			OR	NOT bSensAPVorhanden
			AND	NOT bE_sensRP
			AND		fbZeitAP.Q
			
			OR		bSensAPVorhanden
			AND NOT bSensRPVorhanden
			AND		bE_sensAP
			
			OR		bSensAPVorhanden
			AND		bE_sensAP
			AND NOT bE_sensRP) THEN
			
	eStatus := AktorStatus.inAP;
	
	IF			(eAnfrage = AktorStatus.zuAP) THEN
		bFalschePos := FALSE;
		eAnfrage := AktorStatus.default;
	END_IF

//http://www.32x8.com/sop6_____A-B-C-D-E-F_____m_1-3-5-7-10-11-14-15-17-19-26-27___________option-0_____989781966178824394701
ELSIF		NOT bA_arbeitsPos
		AND (NOT bSensAPVorhanden
		AND NOT bSensRPVorhanden
		AND		fbZeitRP.Q
		
		OR	NOT bSensRPVorhanden
		AND NOT bE_sensAP
		AND		fbZeitRP.Q
		
		OR	NOT bSensAPVorhanden
		AND		bSensRPVorhanden
		AND		bE_sensRP
		
		OR		bSensRPVorhanden
		AND NOT bE_sensAP
		AND		bE_sensRP) THEN
		
	eStatus := AktorStatus.inRP;
	
	IF			(eAnfrage = AktorStatus.zuRP) THEN
		bFalschePos := FALSE;
		eAnfrage := AktorStatus.default;
	END_IF
ELSE
	eStatus := AktorStatus.default;
END_IF

//Nothalt
IF		NOT	MAIN.bE_NotHalt THEN
	bArbeitsPos := FALSE;
	bFalschePos := FALSE;
END_IF

//Handbetrieb
IF			MAIN.bE_Handbetrieb THEN
	IF			bBtnHandausloesung THEN
		bBtnHandausloesung := FALSE;
		handAusloesung();
	END_IF
ELSE
	bBtnHandausloesung := FALSE;
END_IF

//Positionsüberwachung Handbetrieb
fbFtrigHandbetr(CLK := Main.bE_Handbetrieb);

IF 			(fbFtrigHandbetr.Q
	OR		fbSchrittbetrieb.bSendFalschePosError)
	AND		bFalschePos THEN
	
	IF			bA_arbeitsPos THEN
		EventLogger.aErrorLog[250].ipArguments.Clear().AddString(sBezeichnung).AddString('Ruheposition');
	ELSE
		EventLogger.aErrorLog[250].ipArguments.Clear().AddString(sBezeichnung).AddString('Arbeitsposition');
	END_IF
	
	EventLogger.aErrorLog[250].Send(0);
END_IF

IF 			bFalschePos THEN
	fbSchrittbetrieb.bAktorPosNIO := TRUE;
	Main.bPosNachHbNio := TRUE;
END_IF

METHOD arbeitsPos : BOOL
VAR_INPUT
END_VAR
VAR_INST
	bPrevOutputState: 		BOOL;
END_VAR
VAR
	stSchrittEintrag:		ST_SchrittQueue;
END_VAR
stSchrittEintrag.fbAktor REF= THIS^;	
stSchrittEintrag.bGesetzt := TRUE;

//*************************************************************************************
IF		NOT Main.bE_Handbetrieb 
	AND NOT Main.bProgStop
	OR		bHandOverride

	OR		MAIN.bE_Handbetrieb							//Schritt vorwaerts im Handbetrieb
	AND		fbSchrittbetrieb.bAblaufFreigabe THEN
	
	//*************************************************************************************
	IF		NOT bArbeitsPos THEN	//Beim Wechsel des Ausgangs Bewegung in queue aufnehmen
		fbSchrittbetrieb.addToQueue(stSchrittEintrag);
	END_IF
	//*************************************************************************************
	
	bArbeitsPos := TRUE;
	
ELSIF		MAIN.bE_Handbetrieb		//Wenn im Handbetrieb der Aktor, welcher der Ablauf setzten will, verfahren wird, muss die bewegung in die queue aufgenommen werden
	AND	NOT bPrevOutputState
	AND		bArbeitsPos THEN
	fbSchrittbetrieb.addToQueue(stSchrittEintrag);
END_IF

eAnfrage := AktorStatus.zuAP;
bStartUberpruefung := TRUE;			//Damit erst nach dem ersten Befehl die Fehlermeldungen geschrieben werden (sonst sind alle unten vor den Init Ereignissen geloggt)
bPrevOutputState := bArbeitsPos;

arbeitsPos := 			(eStatus = AktorStatus.inAP)
				OR  	((tZeitAP = T#0S)
				AND NOT bSensAPVorhanden
				AND NOT bSensRPVorhanden
				AND		bArbeitsPos);
END_METHOD

METHOD FB_init : BOOL
VAR_INPUT
	bInitRetains:			 	BOOL; // if TRUE, the retain variables are initialized (warm start / cold start)
	bInCopyCode: 				BOOL;  // if TRUE, the instance afterwards gets moved into the copy code (online change)
	
	bSensAPVorhanden:			BOOL;
	bSensRPVorhanden:			BOOL;
	
	tZeitRP:					TIME := T#2S;
	tZeitAP:					TIME := T#2S;
	
	nErrorIdAP:					INT;
	nErrorIdRP:					INT;
	
	sBezeichnung:				String;			//Bezeichnung für Handbetriebfehlermeldung
END_VAR
THIS^.bSensAPVorhanden	:= bSensAPVorhanden;
THIS^.bSensRPVorhanden	:= bSensRPVorhanden;
THIS^.tZeitRP			:= tZeitRP;
THIS^.tZeitAP			:= tZeitAP;
THIS^.nErrorIdAP		:= nErrorIdAP;
THIS^.nErrorIdRP		:= nErrorIdRP;
THIS^.sBezeichnung		:= sBezeichnung;
END_METHOD

METHOD handAusloesung
VAR_INPUT
END_VAR
bArbeitsPos := NOT bArbeitsPos;

bFalschePos := NOT bFalschePos;
END_METHOD

METHOD inAP : BOOL
VAR_INPUT
END_VAR
inAP := (eStatus = AktorStatus.inAP);
END_METHOD

METHOD inRP : BOOL
VAR_INPUT
END_VAR
inRP := (eStatus = AktorStatus.inRP);
END_METHOD

METHOD ruhePos : BOOL
VAR_INPUT
END_VAR
VAR_INST
	bPrevOutputState: 		BOOL;
END_VAR
VAR
	stSchrittEintrag:		ST_SchrittQueue;
END_VAR
stSchrittEintrag.fbAktor REF= THIS^;

//*************************************************************************************
IF		NOT Main.bE_Handbetrieb 
	AND NOT Main.bProgStop
	OR		bHandOverride

	OR		MAIN.bE_Handbetrieb							//Schritt vorwaerts im Handbetrieb
	AND		fbSchrittbetrieb.bAblaufFreigabe THEN
	
	//*************************************************************************************
	IF			bArbeitsPos THEN	//Beim Wechsel des Ausgangs Bewegung in queue aufnehmen
		fbSchrittbetrieb.addToQueue(stSchrittEintrag);
	END_IF
	//*************************************************************************************
	
	bArbeitsPos := FALSE;
	
ELSIF		MAIN.bE_Handbetrieb		//Wenn im Handbetrieb der Aktor, welcher der Ablauf setzten will, verfahren wird, muss die bewegung in die queue aufgenommen werden
	AND	 	bPrevOutputState
	AND	NOT	bArbeitsPos THEN
	fbSchrittbetrieb.addToQueue(stSchrittEintrag);
END_IF

eAnfrage := AktorStatus.zuRP;
bStartUberpruefung := TRUE;			//Damit erst nach dem ersten Befehl die Fehlermeldungen geschrieben werden (sonst sind alle unten vor den Init Ereignissen geloggt)
bPrevOutputState := bArbeitsPos;

ruhePos  := 		(eStatus = AktorStatus.inRP)
			OR  	((tZeitRP = T#0S)
			AND NOT bSensAPVorhanden
			AND NOT bSensRPVorhanden
			AND	NOT bArbeitsPos);
END_METHOD

METHOD stopUeberpruefung
VAR_INPUT
END_VAR
bStartUberpruefung := FALSE;
END_METHOD

END_FUNCTION_BLOCK

// ---- POUs/EventLogger/EventLogger.TcPOU
PROGRAM EventLogger
VAR
	bInit:			BOOL:=TRUE;
	
	aAlarm:			ARRAY[0..Parameter.cAnzEvents] OF FB_Event;
	aMessage:		ARRAY[0..Parameter.cAnzEvents] OF FB_Event;
	aWarnung:		ARRAY[0..Parameter.cAnzEvents] OF FB_Event;
	aErrorLog:		ARRAY[0..Parameter.cAnzEvents] OF FB_Event;
	
	i:				INT;
	j:				INT;
	
	
	
	fbTime 			: NT_GetTime;
END_VAR
VAR PERSISTENT	
	aLoggedEvents:	ARRAY[0..Parameter.cAnzLoggedEvents] OF ST_EventTabelle;
END_VAR

IF bInit THEN
    bInit := FALSE; 
	//Station 1
	aAlarm[13].setText('error', 'Aktor 1 hat Arbeitsposition nicht erreicht oder verloren');
	aAlarm[14].setText('error', 'Aktor 1 hat Ruheposition nicht erreicht oder verloren');
	aAlarm[15].setText('error', 'Aktor 2 hat Arbeitsposition nicht erreicht oder verloren');
	aAlarm[16].setText('error', 'Aktor 2 hat Ruheposition nicht erreicht oder verloren');
	aAlarm[17].setText('error', 'Aktor 3 hat Arbeitsposition nicht erreicht oder verloren');
	aAlarm[18].setText('error', 'Aktor 3 hat Ruheposition nicht erreicht oder verloren');
	aAlarm[19].setText('error', 'Aktor 4 hat Arbeitsposition nicht erreicht oder verloren');
	aAlarm[20].setText('error', 'Aktor 4 hat Ruheposition nicht erreicht oder verloren');
	aAlarm[21].setText('error', 'Aktor 5 hat Arbeitsposition nicht erreicht oder verloren');
	aAlarm[22].setText('error', 'Aktor 5 hat Ruheposition nicht erreicht oder verloren');
	aAlarm[23].setText('error', 'Aktor 6 hat Arbeitsposition nicht erreicht oder verloren');
	aAlarm[24].setText('error', 'Aktor 6 hat Ruheposition nicht erreicht oder verloren');
	
	aAlarm[39].setText('error', 'Kein Teil in Aufnahme. Station per Reset zurücksetzen');
	aAlarm[40].setText('error', 'Not-Halt muss getestet werden');
	

	//	
	aAlarm[100].setText('error', 'Fehler Safety. Anlage mittels Hauptschalter neu starten');
	
	aAlarm[253].setText('error', 'Es wurde {0} Mal in Folge Ausschuss erkannt. Bitte Fehler beheben und "Stoerung Quittieren" betaetigen');
	aAlarm[257].setText('error', 'Luftdruck ist ausserhalb von 5.0 - 6.0bar');
	//
	
	aAlarm[262].setText('error', 'Informationen konnten nicht an Datenbank gesendet werden. Um erneut zu senden, Störung quittieren');
	aAlarm[264].setText('error', 'Senden an Datenbank nicht möglich. (Queue voll) Bitte an Support wenden');

	//
	aErrorLog[230].setText('error', 'Anlage kann nicht gestartet werden, da der Programmablaufunterbruch aktiv ist');
	aErrorLog[231].setText('error', 'Anlage kann nicht gestartet werden, da sich ein Aktor in der falschen Position befindet (im Handbetrieb verfahren)');
	aErrorLog[232].setText('error', 'Anlage kann nicht gestartet werden, da der Handbetrieb aktiviert ist');
	aErrorLog[233].setText('error', 'Anlage kann nicht gestartet werden, da sie nicht fertig Initialisiert ist');
	aErrorLog[234].setText('error', 'Anlage kann nicht gestartet werden, da kein Artikel vorgewaehlt wurde');
	aErrorLog[235].setText('error', 'Anlage kann nicht gestartet werden, da zu viel Ausschuss in Folge produziert wurde');
	aErrorLog[250].setText('error', '{0} sollte sich in der {1} befinden (Falsche Position beim verlassen des Handbetriebs)');
	//
	aErrorLog[260].setText('error', 'Überstromschutzklemme {0} Kanal {1} {2}');
	aErrorLog[261].setText('error', 'MQTT-Message Timeout. Art: {0}, Kennung: {1}');
	aErrorLog[263].setText('error', 'MQTT-Message Error. Art: {0}, Grund: {1}, Kennung: {2}');
	//
	//
	aErrorLog[300].setText('error', '{0}');
	//
	aWarnung[300].setText('warnung', '{0}');
	//
	aMessage[10].setText('info', 'Init wartet auf {0}');
	aMessage[11].setText('info', 'Init fertig');
	aMessage[300].setText('info', '{0}');
	
	
	FOR i := 0 TO Parameter.cAnzLoggedEvents DO
		IF			aLoggedEvents[i].sStatus = 'Aktiv'
			or		aLoggedEvents[i].bPinned THEN
			aLoggedEvents[i].sStatus := 'Cleared';
			aLoggedEvents[i].bPinned := FALSE;
		END_IF
	END_FOR
END_IF

fbTime(START := TRUE);
fbTime(START := FALSE);

FOR i := 0 TO Parameter.cAnzEvents DO
	aAlarm[i](nID := i);
	aMessage[i](nID := i);
	aWarnung[i](nID := i);
	aErrorLog[i](nID := i);
END_FOR

METHOD logEvent
VAR_INPUT
	nEventId:	INT;
	sText:		STRING(255);
	sSeverity: 	STRING;
	bPin:		BOOL;
END_VAR
VAR
	i:			INT;
END_VAR
FOR i := Parameter.cAnzLoggedEvents-1 TO 0 BY -1 DO
	
	IF 		NOT aLoggedEvents[i].bPinned 		//Nicht gepinnte Events schieben
		OR		bPin THEN						//Gepinnte Events auch schieben falls der neue gepinnt werden soll
		aLoggedEvents[i+1] := aLoggedEvents[i];
	ELSE					
		EXIT;
	END_IF
END_FOR



aLoggedEvents[i+1].bPinned := bPin;
aLoggedEvents[i+1].sText := sText;
aLoggedEvents[i+1].sSeverity := sSeverity;
aLoggedEvents[i+1].nEventId := nEventId;
aLoggedEvents[i+1].sTimestamp := SYSTEMTIME_TO_STRING(fbTime.TIMESTR);

IF			bPin THEN
	aLoggedEvents[i+1].sStatus := 'Aktiv';
ELSE 
	aLoggedEvents[i+1].sStatus := '';
END_IF
END_METHOD

METHOD unpinEvent
VAR_INPUT
	nID:		INT;
END_VAR
FOR i := 0 TO Parameter.cAnzLoggedEvents DO	
	IF 			(aLoggedEvents[i].nEventId = nID)
		AND	 	aLoggedEvents[i].bPinned THEN
		aLoggedEvents[i].sStatus := 'Cleared';
		aLoggedEvents[i].bPinned := FALSE;
	END_IF
END_FOR
END_METHOD

END_PROGRAM

// ---- POUs/EventLogger/FB_Event.TcPOU
FUNCTION_BLOCK FB_Event
VAR_INPUT
	nID:			INT;
	ipArguments:	Tc3_EventLogger.I_TcArguments;
END_VAR
VAR_OUTPUT
END_VAR
VAR
	sText:			STRING(255);
	sSeverity:		STRING;
	
	bInit:			BOOL := TRUE;
	bIsRaised:		BOOL;
	
	
	fbArguments:	FB_Arguments;
END_VAR

ipArguments := fbArguments;

IF			bInit THEN
	bInit := FALSE;
	fbArguments.sOriginalString := sText;
END_IF

fbArguments(sOutText => sText, iInterfacePointer := ipArguments);

PROPERTY bRaised : Bool
GET
bRaised := bIsRaised;
END_GET
END_PROPERTY

METHOD Clear
VAR_INPUT
	a:	INT;
	b: BOOL;

END_VAR
bIsRaised := FALSE;
EventLogger.unpinEvent(nID);
END_METHOD

METHOD Raise
VAR_INPUT
	a:	INT;
END_VAR
bIsRaised := TRUE;
sText := fbArguments.sOutText;
EventLogger.logEvent(nID, sText,sSeverity, TRUE);
END_METHOD

METHOD RequestEventText
VAR_INPUT
	a:	INT;
END_VAR
VAR_IN_OUT
	b:	STRING(255);
END_VAR
VAR_INPUT
	c:	INT;
END_VAR
b := sText;
END_METHOD

METHOD send
VAR_INPUT
	a:	INT;
END_VAR
sText := fbArguments.sOutText;
EventLogger.logEvent(nID, sText,sSeverity, FALSE);
END_METHOD

METHOD setText
VAR_INPUT
	sSeverity:			STRING;
	sText:				STRING(255);
END_VAR
THIS^.sSeverity := sSeverity;
THIS^.sText := sText;
END_METHOD

END_FUNCTION_BLOCK

// ---- POUs/EventLogger/FB_Arguments.TcPOU
FUNCTION_BLOCK FB_Arguments IMPLEMENTS Tc3_EventLogger.I_TcArguments
VAR_INPUT
	sOriginalString:		STRING(255);
	iInterfacePointer:		Tc3_EventLogger.I_TcArguments;
END_VAR
VAR_OUTPUT
	sOutText:				STRING(255);
END_VAR
VAR
	ipArgumentsinterface:	Tc3_EventLogger.I_TcArguments;
	bInit: 					BOOL := TRUE;
END_VAR

IF			bInit THEN
	bInit := FALSE;
	Clear();
END_IF

METHOD AddBlob : Tc3_EventLogger.I_TcArguments
VAR_INPUT
	pData	: Tc3_EventLogger.PVOID;
	cbData	: UINT;
END_VAR
END_METHOD

METHOD AddBool : Tc3_EventLogger.I_TcArguments
VAR_INPUT
	value	: BOOL;
END_VAR
VAR
	sValue:	STRING;
END_VAR
sValue := BOOL_TO_STRING(value);
AddString(sValue);
AddBool := iInterfacePointer;
END_METHOD

METHOD AddByte : Tc3_EventLogger.I_TcArguments
VAR_INPUT
	value	: BYTE;
END_VAR
VAR
	sValue:	STRING;
END_VAR
sValue := (BYTE_TO_STRING(value));
AddString(sValue);
AddByte := iInterfacePointer;
END_METHOD

METHOD AddDInt : Tc3_EventLogger.I_TcArguments
VAR_INPUT
	value	: DINT;
END_VAR
VAR
	sValue:	STRING;
END_VAR
sValue := (DINT_TO_STRING(value));
AddString(sValue);
AddDInt := iInterfacePointer;
END_METHOD

METHOD AddDWord : Tc3_EventLogger.I_TcArguments
VAR_INPUT
	value	: DWORD;
END_VAR
VAR
	sValue:	STRING;
END_VAR
sValue := (DWORD_TO_STRING(value));
AddString(sValue);
AddDWord := iInterfacePointer;
END_METHOD

METHOD AddEventReferenceEx : Tc3_EventLogger.I_TcArguments
VAR_INPUT
	stEventEntry	: Tc3_EventLogger.TcEventEntry;
END_VAR
END_METHOD

METHOD AddEventReferenceId : Tc3_EventLogger.I_TcArguments
VAR_INPUT
	nEventId	: UDINT;
END_VAR
END_METHOD

METHOD AddEventReferenceIdGuid : Tc3_EventLogger.I_TcArguments
VAR_INPUT
	nEventId	: UDINT;
	EventClass	: Tc3_EventLogger.GUID;
END_VAR
END_METHOD

METHOD AddInt : Tc3_EventLogger.I_TcArguments
VAR_INPUT
	value	: INT;
END_VAR
VAR
	sValue:	STRING;
END_VAR
sValue := (INT_TO_STRING(value));
AddString(sValue);
AddInt := iInterfacePointer;
END_METHOD

METHOD AddLInt : Tc3_EventLogger.I_TcArguments
VAR_INPUT
	value	: LINT;
END_VAR
VAR
	sValue:	STRING;
END_VAR
sValue := (LINT_TO_STRING(value));
AddString(sValue);
AddLInt := iInterfacePointer;
END_METHOD

METHOD AddLReal : Tc3_EventLogger.I_TcArguments
VAR_INPUT
	value	: LREAL;
END_VAR
VAR
	sValue:	STRING;
END_VAR
sValue := (LREAL_TO_STRING(value));
AddString(sValue);
AddLReal := iInterfacePointer;
END_METHOD

METHOD AddReal : Tc3_EventLogger.I_TcArguments
VAR_INPUT
	value	: REAL;
END_VAR
VAR
	sValue:	STRING;
END_VAR
sValue := (REAL_TO_STRING(value));
AddString(sValue);
AddReal := iInterfacePointer;
END_METHOD

METHOD AddSInt : Tc3_EventLogger.I_TcArguments
VAR_INPUT
	value	: SINT;
END_VAR
VAR
	sValue:	STRING;
END_VAR
sValue := (SINT_TO_STRING(value));
AddString(sValue);
AddSInt := iInterfacePointer;
END_METHOD

METHOD AddString : Tc3_EventLogger.I_TcArguments
VAR_IN_OUT CONSTANT
	value	: STRING;
END_VAR
VAR
	nPosition:		INT;
END_VAR
nPosition := getNextPlaceholder();
IF			(nPosition > 0) THEN
	sOutText := INSERT(Delete(sOutText, 3, nPosition), value, nPosition-1);
END_IF

AddString := iInterfacePointer;
END_METHOD

METHOD AddStringByValue : Tc3_EventLogger.I_TcArguments
VAR_INPUT
	value	: Tc3_EventLogger.T_MaxString;
END_VAR
END_METHOD

METHOD AddUDInt : Tc3_EventLogger.I_TcArguments
VAR_INPUT
	value	: UDINT;
END_VAR
VAR
	sValue:	STRING;
END_VAR
sValue := (UDINT_TO_STRING(value));
AddString(sValue);
AddUDInt := iInterfacePointer;
END_METHOD

METHOD AddUInt : Tc3_EventLogger.I_TcArguments
VAR_INPUT
	value	: UINT;
END_VAR
VAR
	sValue:	STRING;
END_VAR
sValue := (UINT_TO_STRING(value));
AddString(sValue);
AddUInt := iInterfacePointer;
END_METHOD

METHOD AddULInt : Tc3_EventLogger.I_TcArguments
VAR_INPUT
	value	: ULINT;
END_VAR
VAR
	sValue:	STRING;
END_VAR
sValue := (ULINT_TO_STRING(value));
AddString(sValue);
AddULInt := iInterfacePointer;
END_METHOD

METHOD AddUSInt : Tc3_EventLogger.I_TcArguments
VAR_INPUT
	value	: USINT;
END_VAR
VAR
	sValue:	STRING;
END_VAR
sValue := (USINT_TO_STRING(value));
AddString(sValue);
AddUSInt := iInterfacePointer;
END_METHOD

METHOD AddUtf8EncodedString : Tc3_EventLogger.I_TcArguments
VAR_IN_OUT CONSTANT
	value	: STRING;
END_VAR
END_METHOD

METHOD AddWord : Tc3_EventLogger.I_TcArguments
VAR_INPUT
	value	: WORD;
END_VAR
VAR
	sValue:	STRING;
END_VAR
sValue := (WORD_TO_STRING(value));
AddString(sValue);
AddWord := iInterfacePointer;
END_METHOD

METHOD AddWString : Tc3_EventLogger.I_TcArguments
VAR_IN_OUT CONSTANT
	value	: WSTRING;
END_VAR
END_METHOD

METHOD AddWStringByValue : Tc3_EventLogger.I_TcArguments
VAR_INPUT
	value	: WSTRING(255);
END_VAR
END_METHOD

METHOD Clear : Tc3_EventLogger.I_TcArguments
sOutText := sOriginalString;
Clear := iInterfacePointer;
END_METHOD

METHOD getNextPlaceholder : INT
VAR_INPUT
END_VAR
VAR
	sText:					STRING(255);
	nPosition:				INT;
	nPlaceholder:			INT;
	nNextPlaceholder:		INT := 32767;
	nNextPlaceholderPos:	INT;
	
	nDeleted:				INT;
	
	bNoMorePlaceholders:	BOOL;
END_VAR
sText := sOutText;

REPEAT
	nPosition := FIND(sText, '{');
	
	IF			(nPosition > 0) THEN
		nPlaceholder := STRING_TO_INT(MID(sText, 1, nPosition+1));
		
		IF			(nPlaceholder < nNextPlaceholder) THEN
			nNextPlaceholder := nPlaceholder;
			nNextPlaceholderPos := nPosition+nDeleted;
		END_IF
		
		sText := Delete(sText, nPosition+2, 1);		//Alles bis zum Plazhalter löschen
		nDeleted := nDeleted+nPosition+2;
		
	ELSE
		bNoMorePlaceholders := TRUE;
	END_IF
	
UNTIL 
	bNoMorePlaceholders
END_REPEAT

getNextPlaceholder := nNextPlaceholderPos;
END_METHOD

PROPERTY ipData : Tc3_EventLogger.ITcArguments
GET
END_GET
END_PROPERTY

PROPERTY nCount : UDINT
GET
END_GET
END_PROPERTY

END_FUNCTION_BLOCK

// ---- POUs/FB_Handheld.TcPOU
FUNCTION_BLOCK FB_Handheld
VAR_INPUT
END_VAR
VAR_OUTPUT
	fbVorTrig:				R_TRIG;
	fbZurueckTrig:			R_TRIG;
	nGewaehlteStation:		INT;
END_VAR
VAR
	bE_TasteVor				AT%I*:	BOOL;
	bE_TasteZurueck			AT%I*:	BOOL;
	bE_Zustimmtaster		AT%I*:	BOOL;
	
	bA_LampeHandheld		AT%Q*:	BOOL;
END_VAR

//********************************************************************************
//Handheld
fbVorTrig(CLK := bE_TasteVor AND bE_Zustimmtaster);
fbZurueckTrig(CLK := bE_TasteZurueck AND bE_Zustimmtaster);

bA_LampeHandheld := bE_Zustimmtaster AND MAIN.bE_Handbetrieb;

END_FUNCTION_BLOCK

// ---- POUs/FB_Zykluszeit.TcPOU
FUNCTION_BLOCK FB_Zykluszeit
VAR_INPUT
	bStart:					BOOL;
	fZyklusZeitTask:		REAL;
END_VAR

VAR_OUTPUT
	fZyklusZeit:			REAL;
END_VAR

VAR
	fZykluszaehler:			REAL;
	fZykluszeitTemp:		REAL;
	fbStartFlanke:			R_TRIG;
	fbStopFlanke:			R_TRIG;
	bZyklusMessungAkt:		BOOL;
END_VAR

fbStartFlanke(CLK := bStart);
fbStopFlanke(CLK := NOT bStart);
fZykluszeitTemp := fZykluszaehler * (fZyklusZeitTask/1000);

IF fbStartFlanke.Q THEN
	fZykluszaehler := 0;
	fZyklusZeit := fZykluszeitTemp;
	bZyklusMessungAkt := FALSE;
END_IF

IF			fbStartFlanke.Q 
	AND NOT	bZyklusMessungAkt THEN
	bZyklusMessungAkt := TRUE;
END_IF

IF 		bZyklusMessungAkt THEN
	fZykluszaehler := fZykluszaehler + 1;
END_IF

IF			fbStopFlanke.Q 
	AND 	bZyklusMessungAkt THEN
	bZyklusMessungAkt := FALSE;
END_IF

(*
fbStartFlanke(CLK := bStart);
fbStopFlanke(CLK := bStop);
fZykluszeitTemp := fZykluszaehler * (fZyklusZeitTask/1000);

IF fbStartFlanke.Q THEN
	fZykluszaehler := 0;
	fZyklusZeit := fZykluszeitTemp;
	bZyklusMessungAkt := FALSE;
END_IF

IF			fbStartFlanke.Q 
	AND NOT	bZyklusMessungAkt THEN
	bZyklusMessungAkt := TRUE;
END_IF

IF 		bZyklusMessungAkt
	AND	MAIN.bProduzieren THEN
	fZykluszaehler := fZykluszaehler + 1;
END_IF

IF			fbStopFlanke.Q 
	AND 	bZyklusMessungAkt THEN
	bZyklusMessungAkt := FALSE;
END_IF
*)

END_FUNCTION_BLOCK

// ---- POUs/FB_EL9227.TcPOU
FUNCTION_BLOCK FB_EL9227
VAR_INPUT
		sBezeichnung:	STRING;							// Klemmenbezeichnung
END_VAR
VAR_OUTPUT
		bStoerung:		BOOL;
		stKanal:		ARRAY[1..2] OF ST_EL9227_IN;
		fCurrent:		ARRAY[1..2] OF REAL;			// Umrechunung in A		[1 = 0.01A]
		fVoltageIn:		ARRAY[1..2] OF REAL;			// Umrechunung in V		[1 = 0.1V]
		fVoltageOut:	ARRAY[1..2] OF REAL;			// Umrechunung in V		[1 = 0.1V]
END_VAR
VAR
		nErrorId:		INT;
		sKanal:			ARRAY[1..2] OF STRING;						// String mit Kanalnummer für Fehlermeldung
		i:				INT;
		fbTrig:			ARRAY[1..2] OF F_TRIG;
END_VAR


//***********************************************************************************************
//Fehlermeldung  ==> Aufbau des Fehlertext: Überstromschutzklemme "180A0" Kanal "1" "Kurzschluss"
sKanal[1] := '1 ';
sKanal[2] := '2 ';

FOR i := 1 TO 2 DO
	
	fbTrig[i](CLK := stKanal[i].stStatus.bEnabled);
	
	//FOR i := 1 TO 2 DO
	IF 			fbTrig[i].Q THEN
		//Kurzschluss
		IF		stKanal[i].stStatus.bShortCircuit THEN
			EventLogger.aErrorLog[nErrorId].ipArguments.Clear().AddString(sBezeichnung).AddString(sKanal[i]).AddString('Kurzschluss');		
			
		//Überlast
		ELSIF		stKanal[i].stStatus.bOverload THEN
			EventLogger.aErrorLog[nErrorId].ipArguments.Clear().AddString(sBezeichnung).AddString(sKanal[i]).AddString('Überlast');		
			
		//Hardwareschutz
		ELSIF		stKanal[i].stStatus.bHardwareProtection  THEN
			EventLogger.aErrorLog[nErrorId].ipArguments.Clear().AddString(sBezeichnung).AddString(sKanal[i]).AddString('Hardwareschutz ausgelöst');		
			
		//Überspannung
		ELSIF		stKanal[i].stStatus.bOvervoltage THEN
			EventLogger.aErrorLog[nErrorId].ipArguments.Clear().AddString(sBezeichnung).AddString(sKanal[i]).AddString('Überspannung');		
			
		//Unterspannung
		ELSIF		stKanal[i].stStatus.bUndervoltage THEN
			EventLogger.aErrorLog[nErrorId].ipArguments.Clear().AddString(sBezeichnung).AddString(sKanal[i]).AddString('Unterspannung');		
			
		//Kanal ausgeschaltet durch Taster
		ELSIF		stKanal[i].stStatus.bDisabledBySwitch THEN
			EventLogger.aErrorLog[nErrorId].ipArguments.Clear().AddString(sBezeichnung).AddString(sKanal[i]).AddString('ausgeschaltet durch Taster');
	
		//Kanal ausgeschaltet durch Ausgang
		ELSIF		stKanal[i].stStatus.bDisabledByOutput THEN
			EventLogger.aErrorLog[nErrorId].ipArguments.Clear().AddString(sBezeichnung).AddString(sKanal[i]).AddString('ausgeschaltet durch Ausgang');		
			
		END_IF
		EventLogger.aErrorLog[nErrorId].Send(0);
	END_IF	
	
	fCurrent[i] 	:= INT_TO_REAL(stKanal[i].nCurrent)		/	100;
	fVoltageIn[i] 	:= INT_TO_REAL(stKanal[i].nVoltageIn)	/	10;
	fVoltageOut[i] 	:= INT_TO_REAL(stKanal[i].nVoltageOut)	/	10;
	
	
END_FOR

IF			stKanal[1].stStatus.bEnabled
	AND		stKanal[2].stStatus.bEnabled THEN
	bStoerung := FALSE;	
ELSE
	bStoerung := TRUE;	
END_IF

METHOD FB_init : BOOL
VAR_INPUT
	bInitRetains : BOOL; // if TRUE, the retain variables are initialized (warm start / cold start)
	bInCopyCode : BOOL;  // if TRUE, the instance afterwards gets moved into the copy code (online change)
	
	nErrorId:		INT;
	sBezeichnung:	STRING;	
END_VAR
THIS^.nErrorId		:= nErrorId;
THIS^.sBezeichnung	:= sBezeichnung;
END_METHOD

END_FUNCTION_BLOCK

// ---- POUs/FB_Stundenleistung.TcPOU
FUNCTION_BLOCK FB_Stundenleistung
VAR_INPUT
	fZyklusZeitTask: 		REAL;
	bProduzieren:			BOOL;
	nStueckZaehlerAnlage:	UDINT;		
	bInitBeendet:			BOOL;
END_VAR

VAR_OUTPUT
	fStundenLeistung:		REAL;
END_VAR

VAR
	fZykluszaehler:			REAL;
	fAktZaehler:			REAL;
	bAktualisieren:			BOOL;
	fbFlankeInit:			R_TRIG;
	nStueckzaehlerStart:	UDINT;
	nStueckZahlBerechnet:	UDINT;
	
END_VAR

// Nach Init aktuellen Zählerstand abspeichern
fbFlankeInit(CLK:=bInitBeendet);
IF			fbFlankeInit.Q THEN
	nStueckzaehlerStart := nStueckZaehlerAnlage;
	fAktZaehler := 0;
END_IF

// Zählerstand rechnen
nStueckZahlBerechnet := nStueckZaehlerAnlage - nStueckzaehlerStart;


IF bProduzieren THEN
	IF			Parameter.cAktRateStundenLeistung <= fZykluszaehler * (fZyklusZeitTask/1000) THEN
		bAktualisieren := TRUE;
		fZykluszaehler := 0;
		fAktZaehler := fAktZaehler + 1;
	ELSE
		bAktualisieren := FALSE;
		fZykluszaehler := fZykluszaehler + 1;
	END_IF
END_IF


IF			Parameter.cAktRateStundenLeistung 	> 0
	AND		fAktZaehler > 0 
	AND		bAktualisieren	THEN
	fStundenLeistung := UDINT_TO_REAL(nStueckZahlBerechnet) / ((Parameter.cAktRateStundenLeistung * fAktZaehler)/3600);
END_IF

END_FUNCTION_BLOCK

// ---- POUs/FB_Wartung.TcPOU
FUNCTION_BLOCK FB_Wartung
VAR_INPUT
END_VAR
VAR_OUTPUT
END_VAR
VAR
	bWartungAnstehend:			BOOL;	

	i:							INT;
	fZeitBisWartung:			LREAL;	
END_VAR
VAR PERSISTENT
	aWartungen:					ARRAY[1..Parameter.cAnzWartungen] OF ST_Wartung;
END_VAR

bWartungAnstehend := FALSE;
FOR i := 1 TO Parameter.cAnzWartungen DO
	
	//***************************************************************************************************
	//Konfiguration übernehmen
	aWartungen[i].sBezeichnung		:= Parameter.aWartungenConfig[i].sBezeichnung;	
	aWartungen[i].sPerson			:= Parameter.aWartungenConfig[i].sPerson;
	aWartungen[i].nZyklenBisWartung	:= Parameter.aWartungenConfig[i].nZyklenBisWartung;
	aWartungen[i].fZeitBisWartung	:= Parameter.aWartungenConfig[i].fZeitBisWartung;
	
	//***************************************************************************************************
	fZeitBisWartung := aWartungen[i].fZeitBisWartung * 3600000;
	
	//Zyklus Zeit hochzählen
	aWartungen[i].fZeitSeitWartung := aWartungen[i].fZeitSeitWartung + Parameter.fZyklusZeitTask;
	
	//Verbleibende Zeit
	IF			(fZeitBisWartung > 0) THEN
//		IF			(fZeitBisWartung - aWartungen[i].fZeitSeitWartung) <= 0 THEN
//			aWartungen[i].sVerbleibendeZeit := 'Abgelaufen';
//		ELSE
			aWartungen[i].sVerbleibendeZeit := LREAL_TO_STRING(LINT_TO_LREAL(LREAL_TO_LINT((fZeitBisWartung - aWartungen[i].fZeitSeitWartung)/36000))/100);
//		END_IF
		aWartungen[i].sZeitBisWartung := REAL_TO_STRING(aWartungen[i].fZeitBisWartung);
	ELSE
		aWartungen[i].sVerbleibendeZeit := '-';
		aWartungen[i].sZeitBisWartung := '-';
	END_IF
	
	//Verbleibende Zyklen
	IF			(aWartungen[i].nZyklenBisWartung > 0) THEN
		IF			(aWartungen[i].nZyklenBisWartung - aWartungen[i].nZyklenSeitWartung) <= 0 THEN
			aWartungen[i].sVerbleibendeZyklen := 'Abgelaufen';
		ELSE
			aWartungen[i].sVerbleibendeZyklen := LINT_TO_STRING(aWartungen[i].nZyklenBisWartung - aWartungen[i].nZyklenSeitWartung);
		END_IF
		aWartungen[i].sZyklenBisWartung := LINT_TO_STRING(aWartungen[i].nZyklenBisWartung);
	ELSE
		aWartungen[i].sVerbleibendeZyklen := '-';
		aWartungen[i].sZyklenBisWartung := '-';
	END_IF

	//***************************************************************************************************
	//Überprüfung ob Wartung ansteht
	aWartungen[i].bAnstehend := 		aWartungen[i].nZyklenSeitWartung >= aWartungen[i].nZyklenBisWartung
								AND		aWartungen[i].nZyklenBisWartung > 0
								
								OR		aWartungen[i].fZeitSeitWartung >= fZeitBisWartung
								AND		aWartungen[i].fZeitBisWartung > 0;
								
	IF			aWartungen[i].bAnstehend THEN
		bWartungAnstehend := TRUE;
	END_IF
	
	//***************************************************************************************************
	//Zurücksetzen
	IF			aWartungen[i].bBtnReset THEN
		aWartungen[i].bBtnReset := FALSE;
		aWartungen[i].fZeitSeitWartung := 0;
		aWartungen[i].nZyklenSeitWartung := 0;
	END_IF
END_FOR

METHOD zyklusHinzufuegen
VAR_INPUT
	eWartung:		Wartungen;
END_VAR
aWartungen[eWartung].nZyklenSeitWartung := aWartungen[eWartung].nZyklenSeitWartung + 1;
END_METHOD

END_FUNCTION_BLOCK

// ---- POUs/FB_Output.TcPOU
FUNCTION_BLOCK FB_Output
VAR_INPUT
	bHandOverride:				BOOL;			//Wenn true kann der Ausgang auch im Handbetrieb geschrieben werden	
	fbSchrittbetrieb:			REFERENCE TO FB_Schrittbetrieb;
	bSendFalschePosError:		BOOL;
END_VAR
VAR_OUTPUT
	bFalschePos:				BOOL;
END_VAR
VAR
	bA_Output					AT%Q*: BOOL;
END_VAR

METHOD reset : BOOL
VAR_INPUT
END_VAR
VAR
	stSchrittEintrag:		ST_SchrittQueue;
END_VAR
stSchrittEintrag.fbOutput REF= THIS^;

//*************************************************************************************
IF		NOT Main.bE_Handbetrieb 
	AND NOT Main.bProgStop
	OR		bHandOverride

	OR		MAIN.bE_Handbetrieb							//Schritt vorwaerts im Handbetrieb
	AND		fbSchrittbetrieb.bAblaufFreigabe THEN
	
	//*************************************************************************************
	IF		 	bA_Output THEN	//Beim Wechsel des Ausgangs Bewegung in queue aufnehmen
		fbSchrittbetrieb.addToQueue(stSchrittEintrag);
	END_IF
	//*************************************************************************************
	
	bA_Output := FALSE;
	reset := TRUE;
END_IF
END_METHOD

METHOD set : BOOL
VAR_INPUT
END_VAR
VAR
	stSchrittEintrag:		ST_SchrittQueue;
END_VAR
stSchrittEintrag.fbOutput REF= THIS^;	
stSchrittEintrag.bGesetzt := TRUE;

//*************************************************************************************
IF		NOT Main.bE_Handbetrieb 
	AND NOT Main.bProgStop
	OR		bHandOverride

	OR		MAIN.bE_Handbetrieb							//Schritt vorwaerts im Handbetrieb
	AND		fbSchrittbetrieb.bAblaufFreigabe THEN
	
	//*************************************************************************************
	IF		NOT bA_Output THEN	//Beim Wechsel des Ausgangs Bewegung in queue aufnehmen
		fbSchrittbetrieb.addToQueue(stSchrittEintrag);
	END_IF
	//*************************************************************************************
	
	bA_Output := TRUE;
	set := TRUE;
END_IF
END_METHOD

END_FUNCTION_BLOCK

// ---- POUs/StdStationen/FB_StationMitZuf.TcPOU
FUNCTION_BLOCK FB_StationMitZuf EXTENDS FB_Station
VAR_INPUT
	ifTeilHolen:			IF_TeilHolen;
END_VAR
VAR_OUTPUT
END_VAR
VAR
	eHolStatus: 			AblaufStatus := AblaufStatus.bereit;
	eStatusGreifer:			StatusGreifer;
	nTeileZaehler:			INT;	
	nAusschussZaehler:		INT;
END_VAR

//********************************************************************************					
//Schrittbetrieb
fbSchrittbetrieb.eHolStatus := eHolStatus;
fbSchrittbetrieb.bAblaufAktiv := fbSchrittbetrieb.bAblaufAktiv OR nTeileZaehler > 0;

//********************************************************************************					
//Handzyklus (Muss Vor SUPER Call sein, damit diese Version vom Hand Zyklus ausgeführt wird)
//IF			bBtnHandZyklus THEN
//	bBtnHandZyklus := FALSE;
//	
//	IF			stStationInfo.bZyklusFertig
//		AND		bRstInPos
//		AND NOT MAIN.bProduzieren THEN
//		IF			MAIN.hatAufnBeiStJob(stStationInfo.nStationsNr) THEN							//Aufnahme will bearbeitet werden (Teile wurden schon bestellt)
//			ifStation.bearbeitenAnfordern(MAIN.getAufnahmeBeiStation(stStationInfo.nStationsNr));	//Aktuelle Aufnahme wird verwendet
//		ELSE																						//Aufnahme will NICHT bearbeitet werden (Teile müssen bestellt werden)
//			MAIN.vorwahlPseudoaufnahme();
//			ifTeilHolen.holenAnfordern();
//			ifStation.bearbeitenAnfordern(Parameter.cAnzAufnahmen+1);								//Pseudoaufnahme wird verwendet
//		END_IF	
//	END_IF
//END_IF

//********************************************************************************					
//Call Basisklasse
SUPER^(stStationInfo := stStationInfo);

//********************************************************************************					
//Ablauf

IF			stStationInfo.bInitBeendet 
	AND NOT stStationInfo.bReset
	AND NOT fbSchrittbetrieb.bInQueue THEN
	
	IF			nTeileZaehler > 0  THEN
		ifTeilHolen.teilHolen();
	END_IF
END_IF


IF			(nAusschussZaehler > 0)
	AND		(nTeileZaehler > 1
	OR		(nTeileZaehler > 0
	AND		(eHolStatus = AblaufStatus.bereit))) THEN
	nTeileZaehler := nTeileZaehler-1;
	nAusschussZaehler := nAusschussZaehler-1;
END_IF

//********************************************************************************
//Statusanzeige
IF			stStationInfo.bInitBeendet
	AND	NOT	stStationInfo.bReset
	AND NOT stStationInfo.bInit
	AND NOT (eStatusGreifer = StatusGreifer.teilGeholt)
	AND NOT (eStatusGreifer = StatusGreifer.teilAbgelegt) THEN	
	stStationInfo.sStatus := TO_STRING(eHolStatus);
END_IF

METHOD ausschussMelden
VAR_INPUT
END_VAR
nAusschussZaehler := nAusschussZaehler+1;
END_METHOD

METHOD holenAnfordern
VAR_INPUT
END_VAR
nTeileZaehler := nTeileZaehler+1;
END_METHOD

END_FUNCTION_BLOCK

// ---- POUs/StdStationen/FB_StationMitZufUndVer.TcPOU
FUNCTION_BLOCK FB_StationMitZufUndVer EXTENDS FB_StationMitZuf
VAR_INPUT
	ifTeilBereitstellen:		IF_TeilBereitstellen;
END_VAR
VAR_OUTPUT
END_VAR
VAR
	eBereitstellStatus:		AblaufStatus := AblaufStatus.bereit;
	eStatusZuf:				StatusZufuehrung;
	
	nBereitstellZaehler:	INT;
	nAusschussZaehlerBerSt: INT;
END_VAR

//********************************************************************************					
//Schrittbetrieb
fbSchrittbetrieb.eBereitstellStatus := eBereitstellStatus;
fbSchrittbetrieb.bAblaufAktiv := nBereitstellZaehler > 0;

//********************************************************************************					
//Handzyklus (Muss Vor SUPER Call sein, damit diese Version vom Hand Zyklus ausgeführt wird)
//IF			bBtnHandZyklus THEN
//	bBtnHandZyklus := FALSE;
//	
//	IF			stStationInfo.bZyklusFertig
//		AND		bRstInPos
//		AND NOT MAIN.bProduzieren THEN
//		IF			MAIN.hatAufnBeiStJob(stStationInfo.nStationsNr) THEN							//Aufnahme will bearbeitet werden (Teile wurden schon bestellt)
//			ifStation.bearbeitenAnfordern(MAIN.getAufnahmeBeiStation(stStationInfo.nStationsNr));	//Aktuelle Aufnahme wird verwendet
//		ELSE																						//Aufnahme will NICHT bearbeitet werden (Teile müssen bestellt werden)
//			MAIN.vorwahlPseudoaufnahme();
//			ifTeilBereitstellen.holenAnfordern();
//			ifStation.bearbeitenAnfordern(Parameter.cAnzAufnahmen+1);								//Pseudoaufnahme wird verwendet
//		END_IF	
//	END_IF
//END_IF

//********************************************************************************					
//Call Basisklasse
SUPER^(stStationInfo := stStationInfo);

//********************************************************************************					
//Ablauf

IF			stStationInfo.bInitBeendet 
	AND NOT stStationInfo.bReset
	AND NOT fbSchrittbetrieb.bInQueue THEN
	
	IF			nBereitstellZaehler > 0 THEN
		ifTeilBereitstellen.teilBereitstellen();
	END_IF
END_IF

IF			(nAusschussZaehlerBerSt > 0)
	AND		(nBereitstellZaehler > 1
	OR		(nBereitstellZaehler > 0
	AND		(eBereitstellStatus = AblaufStatus.bereit))) THEN
	nBereitstellZaehler := nBereitstellZaehler-1;
	nAusschussZaehlerBerSt := nAusschussZaehlerBerSt-1;
END_IF

METHOD ausschussMelden
VAR_INPUT
END_VAR
SUPER^.ausschussMelden();
nAusschussZaehlerBerSt := nAusschussZaehlerBerSt+1;
END_METHOD

METHOD holenAnfordern
VAR_INPUT
END_VAR
nTeileZaehler := nTeileZaehler+1;
nBereitstellZaehler := nBereitstellZaehler+1;
END_METHOD

END_FUNCTION_BLOCK

// ---- POUs/Tools.TcPOU
PROGRAM Tools
VAR
END_VAR

METHOD inToleranz : BOOL
VAR_INPUT
	fIstwert:		REAL;
	fMin:			REAL;
	fMax:			REAL;
END_VAR
inToleranz := fIstwert >= fMin AND fIstwert <= fMax;
END_METHOD

METHOD runden : REAL
VAR_INPUT
	fInput:			REAL;
	nAnzStellen:	DINT;
END_VAR

VAR
	nZwResultat:	DINT;
END_VAR
nZwResultat := REAL_TO_DINT(fInput*EXPT(10,nAnzStellen+1));
IF 			(nZwResultat MOD 10) >= 5THEN
	nZwResultat := nZwResultat + 10;
END_IF
nZwResultat := nZwResultat / 10;
runden		:= DINT_TO_REAL(nZwResultat)/EXPT(10,nAnzStellen);
END_METHOD

END_PROGRAM

// ---- GlobalTextList.TcGTLO
TEXTLIST GlobalTextList
  595 = '   Fehlermeldung'
  474 = ' Station %d'
  739 = ' vorhadnen'
  808 = ' Vorhanden'
  649 = '%.0f'
  831 = '%.2f'
  683 = '%2.1f'
  395 = '%d'
  348 = '%f'
  651 = '%f.2'
  798 = '%s'
  447 = '%t[ms]'
  340 = '0546.0000 Kontrollvorrichtung\nBR18'
  420 = '0653 BR84 Bolzen- Querfederautomat'
  195 = '0660 Zweihandauslösung'
  256 = '0661 Universalsteuerung'
  1081 = '0661 Zweihandauslösung'
  302 = '1'
  1689 = '10'
  48 = '10.200.30.146'
  170 = '10.200.30.200'
  847 = '10.200.30.201'
  564 = '10.200.30.??'
  192 = '11'
  1549 = '12'
  1632 = '2'
  257 = '3'
  1773 = '4'
  331 = '4024.22'
  299 = '4024.35'
  188 = '4026.13'
  1848 = '5'
  681 = '6'
  601 = '7'
  1308 = '8'
  1183 = '9'
  1344 = '<< Konfig 1'
  634 = 'Aktiviert'
  1095 = 'Aktor 1'
  322 = 'Aktor 2'
  106 = 'Aktor 3'
  166 = 'Aktor 4'
  610 = 'Aktor 5'
  1480 = 'Aktor 6'
  605 = 'Aktor Nr.'
  367 = 'Aktorkonfigurator'
  365 = 'Aktpos:'
  698 = 'Aktuelle Kraft:'
  173 = 'Aktuelle Pos:'
  585 = 'Aktuelle Position:'
  503 = 'Aktuelle Vorwahl:'
  60 = 'Anstehend'
  851 = 'Anz. Zyklen'
  383 = 'Anzeige Station'
  134 = 'Anzeigen'
  145 = 'Artikel:'
  853 = 'Artikeltyp:'
  303 = 'Auftrag:'
  14 = 'Auftragsmenge'
  790 = 'Auftragsmenge:'
  327 = 'Auslauf'
  72 = 'Ausschuss'
  1088 = 'Auswahl Schritt'
  716 = 'Beckhoff CP6606-0001-0020'
  577 = 'Betriebssystem:'
  697 = 'Bewegung ausführen'
  369 = 'Bezeichnung'
  875 = 'Bitte\nDummy\nprüfen'
  362 = 'Bolzen Anschlag Links'
  321 = 'Bolzen Anschlag Rechts'
  735 = 'Bolzen Bahn abblasen Links'
  255 = 'Bolzen Bahn abblasen links'
  283 = 'Bolzen Bahn abblasen Rechts'
  870 = 'Bolzen Entleeren'
  104 = 'Bolzen Vereinz Links'
  280 = 'Bolzen Vereinz Rechts'
  422 = 'Deaktiviert'
  499 = 'Diagnose'
  251 = 'Dummy:'
  613 = 'Durchzuführen von'
  310 = 'Einstellungen'
  344 = 'Ersteller, Datum:'
  308 = 'Event Logger'
  639 = 'Ext. Bereit'
  1322 = 'Ext. Start'
  1015 = 'Fahrzeit [ms]'
  452 = 'Fahrzeit[ms]'
  753 = 'Feder Abblasen Puffer'
  898 = 'Feder Abblasen Topf'
  294 = 'Feder Entstörer'
  650 = 'Feder Vereinzelung'
  253 = 'Fritten'
  691 = 'Fusspedal'
  446 = 'Gesamtzähler:\t         %d'
  386 = 'Gesamtzähler:\t     %d'
  568 = 'Gesamtzähler:\t%d'
  223 = 'Geschwindigkeit:'
  406 = 'Grundposition Anfahren'
  779 = 'Gutteile'
  1191 = 'Haltezeit [ms]'
  184 = 'Handbetrieb'
  990 = 'Hardware:'
  293 = 'Hauptzylinder'
  778 = 'HV'
  964 = 'HV Ausschuss'
  16 = 'Informationen'
  89 = 'IP:'
  957 = 'Ist - Spannung (V)'
  583 = 'Ist:'
  1483 = 'Ja'
  926 = 'Konfig 2 >>'
  1063 = 'Konfiguration'
  725 = 'Kraftlimit:'
  584 = 'LED Strom Schalten (Achtung kann LED zerstören!)'
  1300 = 'Leeren'
  1763 = 'Löschen'
  728 = 'Max. Zyklen'
  375 = 'Motor'
  606 = 'MQTT Auto-Repeat'
  897 = 'MQTT Ignore Error'
  1569 = 'Nein'
  954 = 'Not-Halt austauschen'
  884 = 'Not-Halt getesten'
  2331 = 'Not-Halt getestet'
  1065 = 'Not-Halt in Ordnung'
  628 = 'Not-Halt testen'
  1166 = 'Nächster Status: %s'
  952 = 'PFS, Mai 2022'
  552 = 'PFS, November 2024'
  705 = 'Presse'
  1205 = 'Presse 1 >>'
  624 = 'Presse 2'
  448 = 'Presse 2 >>'
  55 = 'Presszeit'
  118 = 'Presszeit [ms]'
  752 = 'Prisma Abdeckung'
  1744 = 'Programm'
  1294 = 'Programm laden'
  540 = 'Prüfergebnis:'
  609 = 'Reset'
  791 = 'Reset Auftragszähler'
  688 = 'Reset Station'
  561 = 'Reset Station 1'
  876 = 'Reset Station 2'
  1218 = 'Reset Station1'
  854 = 'Reset Station2'
  845 = 'S'
  1056 = 'S%d'
  953 = 'Save Persistent Var'
  911 = 'Schalt-\nfunktion\nNIO'
  50 = 'Schliesser'
  2021 = 'Schritt'
  443 = 'Schritt 1 - 6'
  867 = 'Schritt 7 - 12'
  776 = 'Schrittbetrieb'
  955 = 'Sensor 1'
  1453 = 'Sensor 2'
  228 = 'Sensor 3'
  1224 = 'Sensor 4'
  491 = 'Sensor 5'
  596 = 'Sensor 6'
  986 = 'Sensor 7'
  421 = 'Sensor 8'
  935 = 'Sensor AP'
  472 = 'Sensor Arbeitspo'
  641 = 'Sensor Arbeitspos'
  969 = 'Sensor RP'
  82 = 'Sensor Ruhepos'
  1116 = 'Sensor Teil anwesesen'
  319 = 'Sensor Teil anwesesend'
  942 = 'Sensor Übernahme'
  475 = 'Set'
  1192 = 'Soll - Strom (mA)'
  550 = 'Soll das bestehende Programm\nüberschrieben '
  586 = 'Soll das bestehende Programm\nüberschrieben werden?'
  1133 = 'Soll das bestehende Programm überschrieben '
  83 = 'Soll das bestehende Programmüberschrieben '
  77 = 'Soll Max:'
  239 = 'Soll Min:'
  92 = 'Spannung:'
  189 = 'Speichern'
  835 = 'Speichern Persistent Var'
  2146 = 'Start Taste'
  1949 = 'Starttaste'
  1222 = 'Station'
  441 = 'Station %d'
  1094 = 'Station 1'
  297 = 'Station 1 aktiv'
  1060 = 'Station 2'
  1402 = 'Station 2 aktiv'
  592 = 'Stations-Auswahl'
  504 = 'Status Montagestation:'
  844 = 'Status:'
  401 = 'Status: %s'
  1137 = 'Störung\nQuittieren'
  247 = 'Stückzähler Auftrag:'
  235 = 'Stückzähler Gesamt:'
  320 = 'Stückzähler Tag:'
  878 = 'Teil anw.'
  476 = 'Teil anwesend'
  1 = 'TwinCAT Version:'
  1266 = 'Typ'
  1010 = 'Verbl. Zeit (h)'
  1536 = 'Verbl. Zyklen'
  1456 = 'Verbleibende Zeit (h)'
  159 = 'Verbleibende Zyklen'
  663 = 'Vorhanden'
  423 = 'Vorrichtung:'
  771 = 'Vorwahl:'
  473 = 'VV'
  187 = 'Wartung'
  1756 = 'Wechselbetrieb'
  300 = 'Widerstand (mOhm)'
  836 = 'Widerstand messen'
  392 = 'Widerstand:'
  518 = 'Windows 7.00 Embedded'
  1523 = 'WYR, April2025'
  138 = 'WYR, Mai 2025'
  2078 = 'WYR, Mai2025'
  498 = 'WYR, März 2025'
  391 = 'Zange'
  539 = 'Zeit bis Wart. (h)'
  178 = 'Zeit bis Wartung (h)'
  709 = 'Zeit [ms]'
  135 = 'Zielpos:'
  65 = 'Zielposition:'
  645 = 'Zurück'
  560 = 'Zusatzzylinder'
  814 = 'Zusatzzylinder 01'
  381 = 'Zusatzzylinder 02'
  615 = 'Zusatzzylinder 1 vorhadnen'
  261 = 'Zweihand-Schalter austauschen'
  222 = 'Zykl. bis Wart.'
  551 = 'Zyklen bis Wartung'
  109 = 'Zyklusbetrieb'
  617 = 'Zykluszeit:'
  940 = 'Öffner'
END_TEXTLIST

// ---- VISUs/Konfig2.TcVIS
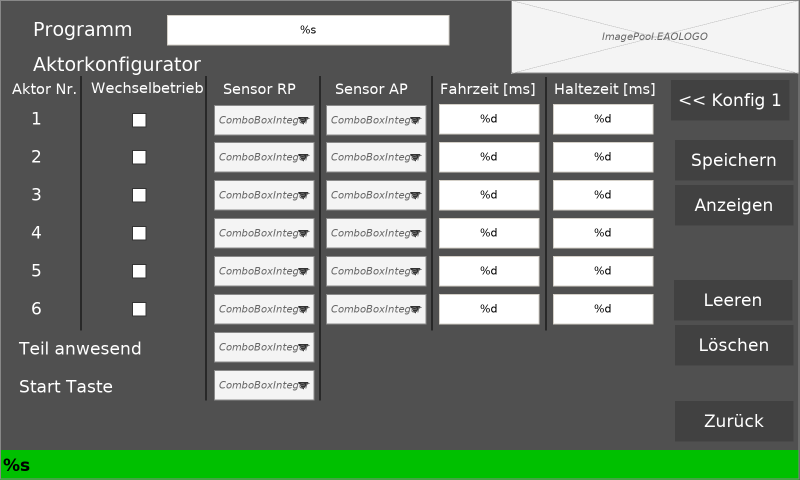
VISUALIZATION Konfig2  // 800x480
    Image (511,0 288x73), image: ImagePool.EAOLOGO
    Textfield (30,15 200x29), "Programm"
    Rectangle (0,450 799x30), "%s", text variable: MAIN.HMI.sStatus, colour variable: MAIN.HMI.nColorInfoBalken
        p3450524324: MAIN.HMI.nColorInfoBalken
    Textfield (220,74 109x30), "Sensor RP"
    Textfield (332,74 109x30), "Sensor AP"
    RoundedRectangle (675,325 118x40), "Löschen"
        OnMouseClick: execute { MAIN.HMI.bBtnProgrammLoeschen := TRUE; }
    Textfield (9,74 73x30), "Aktor Nr."
    Line (206,400) (206,76)
    Line (320,400) (320,76)
    Line (432,330) (432,76)
    Textfield (437,74 109x30), "Fahrzeit [ms]"
    Line (546,330) (546,77)
    Textfield (167,15 282x30), "%s", text variable: MAIN.HMI.ProgrammTemp.sName
        OnMouseClick: write the text variable via VisuDialogs.Keypad
    Textfield (551,74 109x30), "Haltezeit [ms]"
    RoundedRectangle (675,140 118x40), "Speichern", colour toggle: MAIN.fbWritePersistentData.BUSY
        OnMouseClick: execute { MAIN.HMI.bBtnProgrammSpeichern := TRUE; }
    RoundedRectangle (675,185 118x40), "Anzeigen"
        OnMouseClick: execute { MAIN.HMI.bBtnProgrammAnzeigen := TRUE; }
    Textfield (30,50 200x29), "Aktorkonfigurator"
    RoundedRectangle (671,80 118x40), "<< Konfig 1"
        OnMouseClick: change screen: Konfig1
    RoundedRectangle (2011,204 118x40), "<< Konfig 1", colour toggle: MAIN.fbWritePersistentData.BUSY
        OnMouseClick: execute { MAIN.HMI.bBtnProgrammSpeichern := TRUE; }
    Textfield (28,104 34x29), "1"
    Textfield (28,180 34x29), "3"
    Textfield (28,218 34x29), "4"
    Textfield (28,142 34x29), "2"
    Textfield (28,256 34x29), "5"
    Textfield (28,294 34x29), "6"
    Textfield (439,104 100x30), "%d", text variable: MAIN.HMI.ProgrammTemp.aAktorKonfig[1].nFahrZeit
        OnMouseClick: write the text variable via VisuDialogs.Numpad
    Textfield (553,104 100x30), "%d", text variable: MAIN.HMI.ProgrammTemp.aAktorKonfig[1].nHalteZeit
        OnMouseClick: write the text variable via VisuDialogs.Numpad
    Textfield (439,142 100x30), "%d", text variable: MAIN.HMI.ProgrammTemp.aAktorKonfig[2].nFahrZeit
        OnMouseClick: write the text variable via VisuDialogs.Numpad
    Textfield (553,142 100x30), "%d", text variable: MAIN.HMI.ProgrammTemp.aAktorKonfig[2].nHalteZeit
        OnMouseClick: write the text variable via VisuDialogs.Numpad
    Textfield (439,180 100x30), "%d", text variable: MAIN.HMI.ProgrammTemp.aAktorKonfig[3].nFahrZeit
        OnMouseClick: write the text variable via VisuDialogs.Numpad
    Textfield (553,180 100x30), "%d", text variable: MAIN.HMI.ProgrammTemp.aAktorKonfig[3].nHalteZeit
        OnMouseClick: write the text variable via VisuDialogs.Numpad
    Textfield (439,218 100x30), "%d", text variable: MAIN.HMI.ProgrammTemp.aAktorKonfig[4].nFahrZeit
        OnMouseClick: write the text variable via VisuDialogs.Numpad
    Textfield (553,218 100x30), "%d", text variable: MAIN.HMI.ProgrammTemp.aAktorKonfig[4].nHalteZeit
        OnMouseClick: write the text variable via VisuDialogs.Numpad
    Textfield (439,256 100x30), "%d", text variable: MAIN.HMI.ProgrammTemp.aAktorKonfig[5].nFahrZeit
        OnMouseClick: write the text variable via VisuDialogs.Numpad
    Textfield (553,256 100x30), "%d", text variable: MAIN.HMI.ProgrammTemp.aAktorKonfig[5].nHalteZeit
        OnMouseClick: write the text variable via VisuDialogs.Numpad
    Textfield (439,294 100x30), "%d", text variable: MAIN.HMI.ProgrammTemp.aAktorKonfig[6].nFahrZeit
        OnMouseClick: write the text variable via VisuDialogs.Numpad
    Textfield (553,294 100x30), "%d", text variable: MAIN.HMI.ProgrammTemp.aAktorKonfig[6].nHalteZeit
        OnMouseClick: write the text variable via VisuDialogs.Numpad
    ComboBoxInteger (214,105 100x30), variable: MAIN.HMI.ProgrammTemp.aAktorKonfig[1].nSensRuhePos
    ComboBoxInteger (326,105 100x30), variable: MAIN.HMI.ProgrammTemp.aAktorKonfig[1].nSensArbeitsPos
    Textfield (16,334 143x29), "Teil anwesend"
    ComboBoxInteger (214,332 100x30), variable: MAIN.HMI.ProgrammTemp.nTeilAnw
    ComboBoxInteger (214,142 100x30), variable: MAIN.HMI.ProgrammTemp.aAktorKonfig[2].nSensRuhePos
    ComboBoxInteger (326,142 100x30), variable: MAIN.HMI.ProgrammTemp.aAktorKonfig[2].nSensArbeitsPos
    ComboBoxInteger (214,180 100x30), variable: MAIN.HMI.ProgrammTemp.aAktorKonfig[3].nSensRuhePos
    ComboBoxInteger (326,180 100x30), variable: MAIN.HMI.ProgrammTemp.aAktorKonfig[3].nSensArbeitsPos
    ComboBoxInteger (214,218 100x30), variable: MAIN.HMI.ProgrammTemp.aAktorKonfig[4].nSensRuhePos
    ComboBoxInteger (326,218 100x30), variable: MAIN.HMI.ProgrammTemp.aAktorKonfig[4].nSensArbeitsPos
    ComboBoxInteger (214,256 100x30), variable: MAIN.HMI.ProgrammTemp.aAktorKonfig[5].nSensRuhePos
    ComboBoxInteger (326,256 100x30), variable: MAIN.HMI.ProgrammTemp.aAktorKonfig[5].nSensArbeitsPos
    ComboBoxInteger (214,294 100x30), variable: MAIN.HMI.ProgrammTemp.aAktorKonfig[6].nSensRuhePos
    ComboBoxInteger (326,294 100x30), variable: MAIN.HMI.ProgrammTemp.aAktorKonfig[6].nSensArbeitsPos
    Textfield (16,372 143x29), "Start Taste"
    ComboBoxInteger (214,370 100x30), variable: MAIN.HMI.ProgrammTemp.nFussschalterAktiv, text list: 'TL_JaNein'
    Checkbox (130,105 32x30), variable: MAIN.HMI.ProgrammTemp.aAktorKonfig[1].bReversierBetrieb
    RoundedRectangle (675,401 118x40), "Zurück"
        OnMouseClick: change screen: Zyklusbetrieb
    RoundedRectangle (674,280 118x40), "Leeren"
        OnMouseClick: execute { MAIN.HMI.bBtnKonfigLeeren := TRUE; }
    Checkbox (130,142 32x30), variable: MAIN.HMI.ProgrammTemp.aAktorKonfig[2].bReversierBetrieb
    Checkbox (130,180 32x30), variable: MAIN.HMI.ProgrammTemp.aAktorKonfig[3].bReversierBetrieb
    Checkbox (130,218 32x30), variable: MAIN.HMI.ProgrammTemp.aAktorKonfig[4].bReversierBetrieb
    Checkbox (130,256 32x30), variable: MAIN.HMI.ProgrammTemp.aAktorKonfig[5].bReversierBetrieb
    Checkbox (130,294 32x30), variable: MAIN.HMI.ProgrammTemp.aAktorKonfig[6].bReversierBetrieb
    Textfield (88,73 120x30), "Wechselbetrieb"
    Line (81,330) (81,76)
    Group (826,90 645x290)
        p3560616238: MAIN.HMI.nPopUpXOffset
        RoundedRectangle (0,0 645x290), "%s", text variable: MAIN.HMI.sPopUpText, colour toggle: MAIN.fbWritePersistentData.BUSY, invisible if: NOT MAIN.HMI.bPopUpAnzeigen
        RoundedRectangle (128,197 118x40), "Ja", colour toggle: MAIN.fbWritePersistentData.BUSY, invisible if: NOT MAIN.HMI.bPopUpAnzeigen
            OnMouseClick: execute { MAIN.HMI.bBtnPopUpJa := TRUE; }
        RoundedRectangle (405,198 118x40), "Nein", colour toggle: MAIN.fbWritePersistentData.BUSY, invisible if: NOT MAIN.HMI.bPopUpAnzeigen
            OnMouseClick: execute { MAIN.HMI.bBtnPopUpNein := TRUE; }
END_VISUALIZATION

// ---- VISUs/TL_Aktoren.TcTLO
TEXTLIST TL_Aktoren
  0 = 'keine Aktion'
  1 = 'Aktor1 Vor'
  2 = 'Aktor1 Zurück'
  3 = 'Aktor2 Vor'
  4 = 'Aktor2 Zurück'
  5 = 'Aktor3 Vor'
  6 = 'Aktor3 Zurück'
  7 = 'Aktor4 Vor'
  8 = 'Aktor4 Zurück'
  9 = 'Aktor5 Vor'
  10 = 'Aktor5 Zurück'
  11 = 'Aktor6 Vor'
  12 = 'Aktor6 Zurück'
  13 = 'teilAnwesend'
  14 = 'Ext. Gerät bereit'
  15 = 'Ext. Gerät starten'
  16 = 'warten'
   = ''
END_TEXTLIST

// ---- VISUs/Diagnose.TcVIS
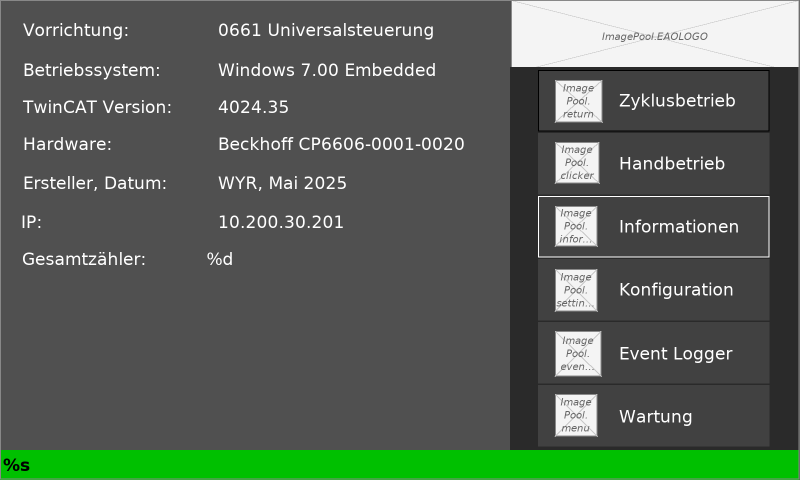
VISUALIZATION Diagnose  // 800x480
    Image (511,0 288x73), image: ImagePool.EAOLOGO
    Rectangle (510,67 289x412)
    Textfield (20,158 177x50), "Ersteller, Datum:"
    Textfield (215,158 288x50), "WYR, Mai 2025"
    Textfield (20,82 177x50), "TwinCAT Version:"
    Textfield (215,82 288x50), "4024.35"
    Textfield (215,45 288x50), "Windows 7.00 Embedded"
    Textfield (20,45 177x50), "Betriebssystem:"
    Textfield (20,5 177x50), "Vorrichtung:"
    Textfield (215,5 288x50), "0661 Universalsteuerung"
    Textfield (20,119 177x50), "Hardware:"
    Textfield (215,119 288x50), "Beckhoff CP6606-0001-0020"
    Textfield (18,197 177x50), "IP:"
    Textfield (215,197 288x50), "10.200.30.201"
    Rectangle (0,450 799x30), "%s", text variable: MAIN.HMI.sStatus, colour variable: MAIN.HMI.nColorInfoBalken
        p3450524324: MAIN.HMI.nColorInfoBalken
    Rectangle (538,70 231x61)
        OnMouseClick: change screen: Zyklusbetrieb
    Textfield (616,70 153x61), "Zyklusbetrieb"
        OnMouseClick: change screen: Zyklusbetrieb
    Rectangle (538,133 231x61)
        OnMouseClick: change screen: Handbetrieb
    Textfield (616,133 153x61), "Handbetrieb"
        OnMouseClick: change screen: Handbetrieb
    Image (555,142 44x41), image: ImagePool.clicker
        OnMouseClick: change screen: Handbetrieb
    Image (555,80 47x42), image: ImagePool.return
        OnMouseClick: change screen: Zyklusbetrieb
    Rectangle (538,196 231x61)
        OnMouseClick: change screen: Diagnose
    Textfield (616,196 153x61), "Informationen"
        OnMouseClick: change screen: Diagnose
    Image (555,206 42x40), image: ImagePool.information
        OnMouseClick: change screen: Diagnose
    Rectangle (538,322 231x61)
        OnMouseClick: change screen: EventLogger
    Textfield (616,323 153x61), "Event Logger"
        OnMouseClick: change screen: EventLogger
    Image (555,331 46x45), image: ImagePool.eventLogger
        OnMouseClick: change screen: EventLogger
    Rectangle (538,259 231x61)
        OnMouseClick: change screen: Konfig1
    Textfield (616,259 153x61), "Konfiguration"
        OnMouseClick: change screen: Konfig1
    Image (555,269 42x42), image: ImagePool.settings
        OnMouseDown: change screen: Konfig1
    Rectangle (538,385 231x61)
        OnMouseClick: change screen: Wartung
    Textfield (616,386 153x61), "Wartung"
        OnMouseClick: change screen: Wartung
    Image (555,394 42x42), image: ImagePool.menu
        OnMouseDown: change screen: Wartung
    Textfield (19,234 477x50), "Gesamtzähler: %d", text variable: MAIN.stStueckzaehler.nGesamt
END_VISUALIZATION

// ---- VISUs/EventLogger.TcVIS
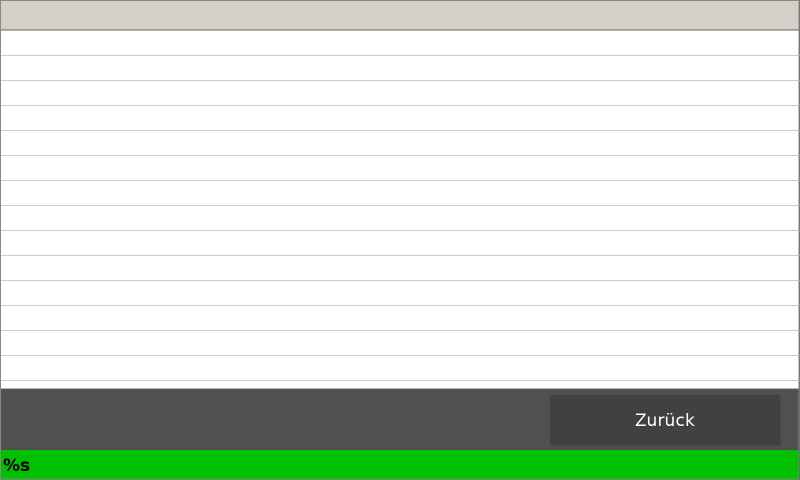
VISUALIZATION EventLogger  // 800x480
    Table (0,0 800x389), data array: EventLogger.aLoggedEvents
        p3854506369: EventLogger.aLoggedEvents[INDEX].sSeverity
        p1892666644: EventLogger.aLoggedEvents[INDEX].sStatus
        p338671338: EventLogger.aLoggedEvents[INDEX].sTimestamp
        p2170511999: EventLogger.aLoggedEvents[INDEX].sText
        p3723444502: EventLogger.aLoggedEvents[INDEX].nEventId
        p1218418051: EventLogger.aLoggedEvents[INDEX].bPinned
        p1755163831: Zeit
        p4092479075: Fehlermeldung
    Rectangle (550,395 230x50), "Zurück"
        OnMouseClick: change screen: Previous Zyklusbetrieb
    Rectangle (0,450 799x30), "%s", text variable: MAIN.HMI.sStatus, colour variable: MAIN.HMI.nColorInfoBalken
        p3450524324: MAIN.HMI.nColorInfoBalken
END_VISUALIZATION

// ---- VISUs/TL_JaNein.TcTLO
TEXTLIST TL_JaNein
  1 = 'Ja'
  0 = 'Nein'
   = ''
END_TEXTLIST

// ---- VISUs/Wartung.TcVIS
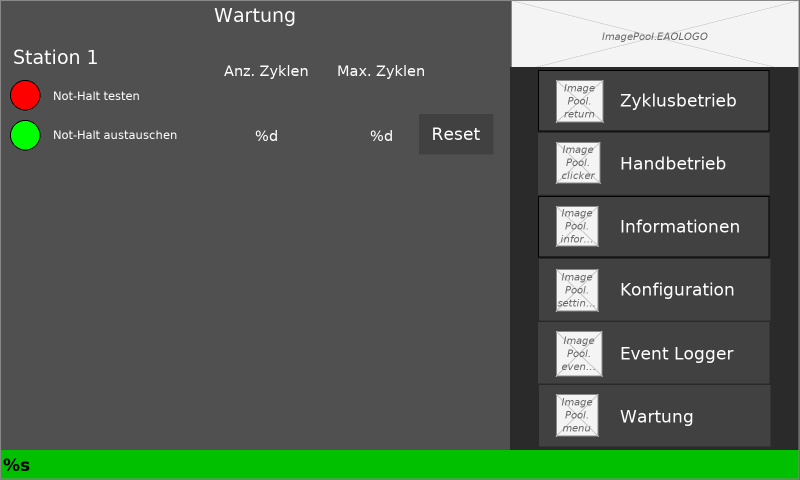
VISUALIZATION Wartung  // 800x480
    Image (511,0 288x73), image: ImagePool.EAOLOGO
    Rectangle (510,67 289x412)
    Textfield (155,1 200x29), "Wartung"
    Rectangle (0,450 799x30), "%s", text variable: MAIN.HMI.sStatus, colour variable: MAIN.HMI.nColorInfoBalken
        p3450524324: MAIN.HMI.nColorInfoBalken
    Rectangle (538,70 231x61)
        OnMouseClick: change screen: Zyklusbetrieb
    Textfield (617,70 153x61), "Zyklusbetrieb"
        OnMouseClick: change screen: Zyklusbetrieb
    Rectangle (538,133 231x61)
        OnMouseClick: change screen: Handbetrieb
    Textfield (617,133 153x61), "Handbetrieb"
        OnMouseClick: change screen: Handbetrieb
    Image (556,142 44x41), image: ImagePool.clicker
        OnMouseClick: change screen: Handbetrieb
    Image (556,80 47x42), image: ImagePool.return
        OnMouseClick: change screen: Zyklusbetrieb
    Rectangle (538,196 231x61)
        OnMouseClick: change screen: Diagnose
    Textfield (617,196 153x61), "Informationen"
        OnMouseClick: change screen: Diagnose
    Image (556,206 42x40), image: ImagePool.information
        OnMouseClick: change screen: Diagnose
    Rectangle (538,322 231x61)
        OnMouseClick: change screen: EventLogger
    Textfield (617,323 153x61), "Event Logger"
        OnMouseClick: change screen: EventLogger
    Image (556,331 46x45), image: ImagePool.eventLogger
        OnMouseClick: change screen: EventLogger
    Rectangle (539,259 231x61)
        OnMouseClick: change screen: Konfig1
    Textfield (617,259 153x61), "Konfiguration"
        OnMouseClick: change screen: Konfig1
    Image (556,269 42x42), image: ImagePool.settings
        OnMouseDown: change screen: Konfig1
    Rectangle (539,385 231x61)
        OnMouseClick: change screen: Wartung
    Textfield (617,386 153x61), "Wartung"
        OnMouseClick: change screen: Wartung
    Image (556,394 42x42), image: ImagePool.menu
        OnMouseDown: change screen: Wartung
    Textfield (50,80 199x32), "Not-Halt testen"
    Textfield (50,120 204x30), "Not-Halt austauschen"
    Ellipse (10,80 30x30), colour toggle: MAIN.fbSt1.bNotHaltTestIO
    Ellipse (10,120 30x30), colour toggle: MAIN.fbSt1.bWarnungNothalt
    Textfield (367,120 78x32), "%d", text variable: Parameter.cMaxZyklNotHalt
    Textfield (252,120 78x32), "%d", text variable: MAIN.fbSt1.nZaehlerNotHalt
    Textfield (221,55 105x32), "Anz. Zyklen"
    Textfield (334,55 105x32), "Max. Zyklen"
    RoundedRectangle (419,114 74x40), "Reset", invisible if: NOT MAIN.fbSt1.bWarnungNothalt
        OnMouseClick: execute { MAIN.fbSt1.bBtnResetWarnNothalt := TRUE; }
    Textfield (10,43 200x29), "Station 1"
END_VISUALIZATION

// ---- VISUs/Handbetrieb.TcVIS
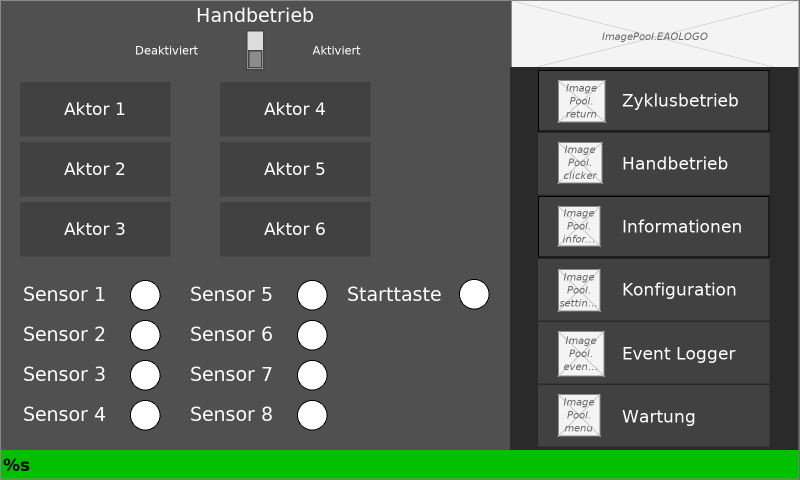
VISUALIZATION Handbetrieb  // 800x480
    Image (511,0 288x73), image: ImagePool.EAOLOGO
    Rectangle (510,67 289x412)
    Textfield (155,1 200x29), "Handbetrieb"
    Textfield (130,25 73x51), "Deaktiviert"
    Textfield (300,25 73x51), "Aktiviert"
    Rectangle (0,450 799x30), "%s", text variable: MAIN.HMI.sStatus, colour variable: MAIN.HMI.nColorInfoBalken
        p3450524324: MAIN.HMI.nColorInfoBalken
    DipSwitch (210,30 90x40), variable: MAIN.bE_Handbetrieb, behaviour: TOGGLE, style: Switch-DipSwitch-Gray
    Textfield (20,82 150x54), "Aktor 1", colour toggle: MAIN.fbSt1.fbAktor[1].bA_arbeitsPos
        OnMouseClick: execute { MAIN.fbSt1.fbAktor[1].bBtnHandausloesung := TRUE; }
    Textfield (20,142 150x54), "Aktor 2", colour toggle: MAIN.fbSt1.fbAktor[2].bA_arbeitsPos
        OnMouseClick: execute { MAIN.fbSt1.fbAktor[2].bBtnHandausloesung := TRUE; }
    Rectangle (538,70 231x61)
        OnMouseClick: change screen: Zyklusbetrieb
    Textfield (619,70 153x61), "Zyklusbetrieb"
        OnMouseClick: change screen: Zyklusbetrieb
    Rectangle (538,133 231x61)
        OnMouseClick: change screen: Handbetrieb
    Textfield (619,133 153x61), "Handbetrieb"
        OnMouseClick: change screen: Handbetrieb
    Image (558,142 44x41), image: ImagePool.clicker
        OnMouseClick: change screen: Handbetrieb
    Image (558,80 47x42), image: ImagePool.return
        OnMouseClick: change screen: Zyklusbetrieb
    Rectangle (538,196 231x61)
        OnMouseClick: change screen: Diagnose
    Textfield (619,196 153x61), "Informationen"
        OnMouseClick: change screen: Diagnose
    Image (558,206 42x40), image: ImagePool.information
        OnMouseClick: change screen: Diagnose
    Rectangle (538,322 231x61)
        OnMouseClick: change screen: EventLogger
    Textfield (619,323 153x61), "Event Logger"
        OnMouseClick: change screen: EventLogger
    Image (558,331 46x45), image: ImagePool.eventLogger
        OnMouseClick: change screen: EventLogger
    Rectangle (538,259 231x61)
        OnMouseClick: change screen: Konfig1
    Textfield (619,259 153x61), "Konfiguration"
        OnMouseClick: change screen: Konfig1
    Image (558,269 42x42), image: ImagePool.settings
        OnMouseDown: change screen: Konfig1
    Rectangle (538,385 231x61)
        OnMouseClick: change screen: Wartung
    Textfield (619,386 153x61), "Wartung"
        OnMouseClick: change screen: Wartung
    Image (558,394 42x42), image: ImagePool.menu
        OnMouseDown: change screen: Wartung
    Textfield (20,202 150x54), "Aktor 3", colour toggle: MAIN.fbSt1.fbAktor[3].bA_arbeitsPos
        OnMouseClick: execute { MAIN.fbSt1.fbAktor[3].bBtnHandausloesung := TRUE; }
    Textfield (220,82 150x54), "Aktor 4", colour toggle: MAIN.fbSt1.fbAktor[4].bA_arbeitsPos
        OnMouseClick: execute { MAIN.fbSt1.fbAktor[4].bBtnHandausloesung := TRUE; }
    Textfield (220,142 150x54), "Aktor 5", colour toggle: MAIN.fbSt1.fbAktor[5].bA_arbeitsPos
        OnMouseClick: execute { MAIN.fbSt1.fbAktor[5].bBtnHandausloesung := TRUE; }
    Textfield (220,202 150x54), "Aktor 6", colour toggle: MAIN.fbSt1.fbAktor[6].bA_arbeitsPos
        OnMouseClick: execute { MAIN.fbSt1.fbAktor[6].bBtnHandausloesung := TRUE; }
    Textfield (20,280 123x29), "Sensor 1"
    Textfield (187,280 123x29), "Sensor 5"
    Textfield (20,320 123x29), "Sensor 2"
    Textfield (187,320 123x29), "Sensor 6"
    Textfield (20,360 123x29), "Sensor 3"
    Textfield (187,360 123x29), "Sensor 7"
    Textfield (187,400 123x29), "Sensor 8"
    Textfield (20,400 123x29), "Sensor 4"
    Ellipse (130,280 30x30), colour toggle: MAIN.fbSt1.bE_Sensor[1]
    Ellipse (130,320 30x30), colour toggle: MAIN.fbSt1.bE_Sensor[2]
    Ellipse (130,360 30x30), colour toggle: MAIN.fbSt1.bE_Sensor[3]
    Ellipse (130,400 30x30), colour toggle: MAIN.fbSt1.bE_Sensor[4]
    Ellipse (297,320 30x30), colour toggle: MAIN.fbSt1.bE_Sensor[6]
    Ellipse (297,280 30x30), colour toggle: MAIN.fbSt1.bE_Sensor[5]
    Ellipse (297,360 30x30), colour toggle: MAIN.fbSt1.bE_Sensor[7]
    Ellipse (297,400 30x30), colour toggle: MAIN.fbSt1.bE_Sensor[8]
    Textfield (344,280 123x29), "Starttaste"
    Ellipse (459,279 30x30), colour toggle: MAIN.bE_Fussschalter
END_VISUALIZATION

// ---- VISUs/Konfig1.TcVIS
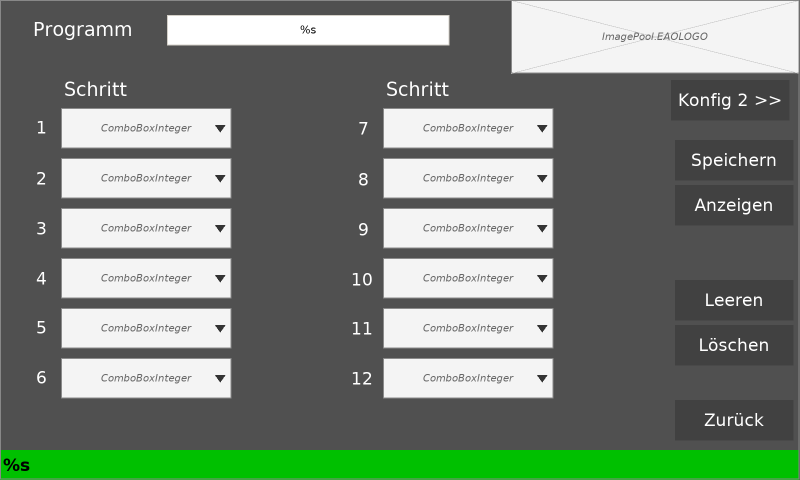
VISUALIZATION Konfig1  // 800x480
    Image (511,0 288x73), image: ImagePool.EAOLOGO
    Textfield (30,15 200x29), "Programm"
    Rectangle (0,450 799x30), "%s", text variable: MAIN.HMI.sStatus, colour variable: MAIN.HMI.nColorInfoBalken
        p3450524324: MAIN.HMI.nColorInfoBalken
    RoundedRectangle (675,325 118x40), "Löschen"
        OnMouseClick: execute { MAIN.HMI.bBtnProgrammLoeschen := TRUE; }
    ComboBoxInteger (61,108 170x40), variable: MAIN.HMI.ProgrammTemp.aAktorBew[1].nNummer, text list: 'TL_Aktoren'
    Textfield (167,15 282x30), "%s", text variable: MAIN.HMI.ProgrammTemp.sName
        OnMouseClick: write the text variable via VisuDialogs.Keypad
    RoundedRectangle (675,140 118x40), "Speichern", colour toggle: MAIN.fbWritePersistentData.BUSY
        OnMouseClick: execute { MAIN.HMI.bBtnProgrammSpeichern := TRUE; }
    RoundedRectangle (675,185 118x40), "Anzeigen"
        OnMouseClick: execute { MAIN.HMI.bBtnProgrammAnzeigen := TRUE; }
    ComboBoxInteger (61,158 170x40), variable: MAIN.HMI.ProgrammTemp.aAktorBew[2].nNummer, text list: 'TL_Aktoren'
    ComboBoxInteger (61,208 170x40), variable: MAIN.HMI.ProgrammTemp.aAktorBew[3].nNummer, text list: 'TL_Aktoren'
    ComboBoxInteger (61,258 170x40), variable: MAIN.HMI.ProgrammTemp.aAktorBew[4].nNummer, text list: 'TL_Aktoren'
    ComboBoxInteger (61,308 170x40), variable: MAIN.HMI.ProgrammTemp.aAktorBew[5].nNummer, text list: 'TL_Aktoren'
    ComboBoxInteger (61,358 170x40), variable: MAIN.HMI.ProgrammTemp.aAktorBew[6].nNummer, text list: 'TL_Aktoren'
    Textfield (61,75 139x29), "Schritt"
    RoundedRectangle (671,80 118x40), "Konfig 2 >>"
        OnMouseClick: change screen: Konfig2
    Textfield (383,75 156x29), "Schritt"
    ComboBoxInteger (383,108 170x40), variable: MAIN.HMI.ProgrammTemp.aAktorBew[7].nNummer, text list: 'TL_Aktoren'
    ComboBoxInteger (383,158 170x40), variable: MAIN.HMI.ProgrammTemp.aAktorBew[8].nNummer, text list: 'TL_Aktoren'
    ComboBoxInteger (383,208 170x40), variable: MAIN.HMI.ProgrammTemp.aAktorBew[9].nNummer, text list: 'TL_Aktoren'
    ComboBoxInteger (383,258 170x40), variable: MAIN.HMI.ProgrammTemp.aAktorBew[10].nNummer, text list: 'TL_Aktoren'
    ComboBoxInteger (383,308 170x40), variable: MAIN.HMI.ProgrammTemp.aAktorBew[11].nNummer, text list: 'TL_Aktoren'
    ComboBoxInteger (383,358 170x40), variable: MAIN.HMI.ProgrammTemp.aAktorBew[12].nNummer, text list: 'TL_Aktoren'
    RoundedRectangle (675,280 118x40), "Leeren"
        OnMouseClick: execute { MAIN.HMI.bBtnKonfigLeeren := TRUE; }
    RoundedRectangle (675,400 118x40), "Zurück"
        OnMouseClick: change screen: Zyklusbetrieb
    Textfield (33,113 34x29), "1"
    Textfield (33,214 34x29), "3"
    Textfield (33,264 34x29), "4"
    Textfield (33,164 34x29), "2"
    Textfield (33,313 34x29), "5"
    Textfield (33,363 34x29), "6"
    Textfield (355,114 34x29), "7"
    Textfield (355,215 34x29), "9"
    Textfield (348,265 34x29), "10"
    Textfield (355,165 34x29), "8"
    Textfield (348,314 34x29), "11"
    Textfield (348,364 34x29), "12"
    Group (800,90 645x290)
        RoundedRectangle (0,0 645x290), "%s", text variable: MAIN.HMI.sPopUpText, colour toggle: MAIN.fbWritePersistentData.BUSY, invisible if: NOT MAIN.HMI.bPopUpAnzeigen
            p3560616238: MAIN.HMI.nPopUpXOffset
        RoundedRectangle (128,197 118x40), "Ja", colour toggle: MAIN.fbWritePersistentData.BUSY, invisible if: NOT MAIN.HMI.bPopUpAnzeigen
            p3560616238: MAIN.HMI.nPopUpXOffset
            OnMouseClick: execute { MAIN.HMI.bBtnPopUpJa := TRUE; }
        RoundedRectangle (405,198 118x40), "Nein", colour toggle: MAIN.fbWritePersistentData.BUSY, invisible if: NOT MAIN.HMI.bPopUpAnzeigen
            p3560616238: MAIN.HMI.nPopUpXOffset
            OnMouseClick: execute { MAIN.HMI.bBtnPopUpNein := TRUE; }
END_VISUALIZATION

// ---- VISUs/Zyklusbetrieb.TcVIS
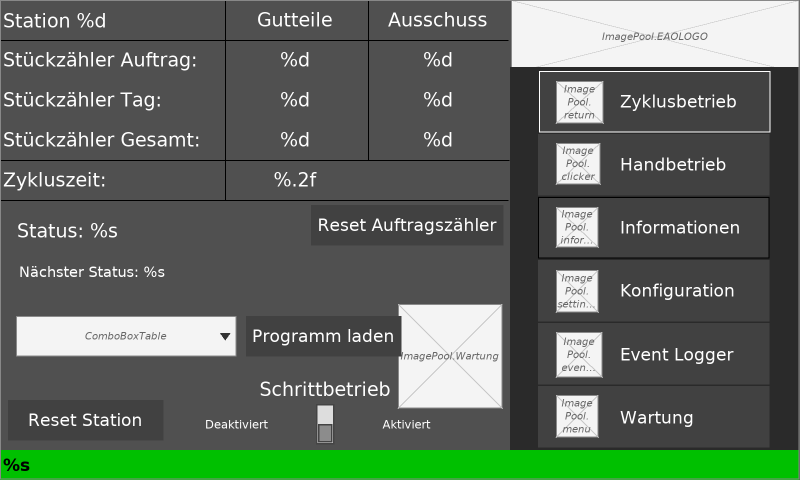
VISUALIZATION Zyklusbetrieb  // 800x480
    Textfield (0,40 225x40), "Stückzähler Auftrag:"
    Image (511,0 288x73), image: ImagePool.EAOLOGO
    Rectangle (510,67 289x412)
    Line (1,160) (509,160)
    Line (225,0) (225,200)
    Line (0,40) (508,40)
    Textfield (0,80 225x40), "Stückzähler Tag:"
    Textfield (0,120 225x40), "Stückzähler Gesamt:"
    Textfield (225,40 140x40), "%d", text variable: MAIN.stStueckzaehler.nGutteileAuftrag
    Line (368,0) (368,160)
    Textfield (225,80 140x40), "%d", text variable: MAIN.stStueckzaehler.nGutteileTag
    Textfield (225,120 140x40), "%d", text variable: MAIN.stStueckzaehler.nGutteileGesamt
    Textfield (368,80 140x40), "%d", text variable: MAIN.stStueckzaehler.nAusschussTag
    Textfield (368,40 140x40), "%d", text variable: MAIN.stStueckzaehler.nAusschussAuftrag
    Textfield (368,120 140x40), "%d", text variable: MAIN.stStueckzaehler.nAusschussGesamt
    Textfield (225,0 140x40), "Gutteile"
    Textfield (368,0 140x40), "Ausschuss"
    Rectangle (0,450 799x30), "%s", text variable: MAIN.HMI.sStatus, colour variable: MAIN.HMI.nColorInfoBalken
        p3450524324: MAIN.HMI.nColorInfoBalken
    Line (0,200) (508,200)
    Textfield (0,160 225x40), "Zykluszeit:"
    Textfield (225,160 140x40), "%.2f", text variable: MAIN.fbZyklusZeitGesamt.fZyklusZeit
    RoundedRectangle (8,400 155x40), "Reset Station"
        OnMouseClick: execute { MAIN.fbSt1.bBtnReset := TRUE; }
    Textfield (0,1 140x40), "Station %d", text variable: MAIN.HMI.nAnzeigeStation
    Textfield (14,211 225x40), "Status: %s", text variable: MAIN.HMI.sStationStatus
    Rectangle (539,71 231x61)
        OnMouseClick: change screen: Zyklusbetrieb
    Textfield (617,71 153x61), "Zyklusbetrieb"
        OnMouseClick: change screen: Zyklusbetrieb
    Rectangle (538,134 231x61)
        OnMouseClick: change screen: Handbetrieb
    Textfield (617,134 153x61), "Handbetrieb"
        OnMouseClick: change screen: Handbetrieb
    Image (556,143 44x41), image: ImagePool.clicker
        OnMouseClick: change screen: Handbetrieb
    Image (556,81 47x42), image: ImagePool.return
        OnMouseClick: change screen: Zyklusbetrieb
    Rectangle (538,197 231x61)
        OnMouseClick: change screen: Diagnose
    Textfield (617,197 153x61), "Informationen"
        OnMouseClick: change screen: Diagnose
    Image (556,207 42x40), image: ImagePool.information
        OnMouseClick: change screen: Diagnose
    Rectangle (538,323 231x61)
        OnMouseClick: change screen: EventLogger
    Textfield (617,324 153x61), "Event Logger"
        OnMouseClick: change screen: EventLogger
    Image (556,332 46x45), image: ImagePool.eventLogger
        OnMouseClick: change screen: EventLogger
    Rectangle (538,260 231x61)
        OnMouseClick: change screen: Konfig1
    Textfield (617,260 153x61), "Konfiguration"
        OnMouseClick: change screen: Konfig1
    Image (556,270 42x42), image: ImagePool.settings
        OnMouseDown: change screen: Konfig1
    Rectangle (538,386 231x61)
        OnMouseClick: change screen: Wartung
    Textfield (617,387 153x61), "Wartung"
        OnMouseClick: change screen: Wartung
    Image (556,395 42x42), image: ImagePool.menu
        OnMouseDown: change screen: Wartung
    Image (398,304 104x104), invisible if: NOT MAIN.fbSt1.bWarnungNothalt, image: ImagePool.Wartung
        OnMouseDown: change screen: Wartung
    RoundedRectangle (311,205 192x40), "Reset Auftragszähler"
        OnMouseClick: execute { MAIN.fbSt1.bBtnResetAuftrZaehler := TRUE; }
    ComboBoxTable (16,316 220x40), variable: MAIN.HMI.nAngewaehltesProg, data array: MAIN.HMI.aProgrammNamen
        p3854506369: MAIN.HMI.aProgrammNamen[INDEX]
        p1892666644: MAIN.HMI.aProgramm[INDEX].sName
        p338671338: MAIN.HMI.aProgramm[INDEX].aAktorBew
        p1128707560: Parameter.cMaxProgramme
    RoundedRectangle (246,316 155x40), "Programm laden", colour toggle: MAIN.HMI.bProgrammGeladen, input disabled if: MAIN.HMI.bProgeammLadenBtnInaktiv
        OnMouseClick: execute { MAIN.HMI.bBtnProgrammLaden := TRUE; }
    Textfield (200,399 73x51), "Deaktiviert"
    Textfield (225,375 200x29), "Schrittbetrieb"
    Textfield (370,399 73x51), "Aktiviert"
    DipSwitch (280,404 90x40), variable: MAIN.HMI.bBtnSchrittbetrieb, behaviour: TOGGLE, style: Switch-DipSwitch-Gray
    Textfield (16,252 225x40), "Nächster Status: %s", text variable: MAIN.fbSt1.sNaechsterSchritt, invisible if: not MAIN.fbSt1.bSchrittbetriebAktiv
END_VISUALIZATION
